// Mitsubishi GX Works2 project: Helloworlddeutrabalho   PLC: Q03UDV

PROGRAM MAIN
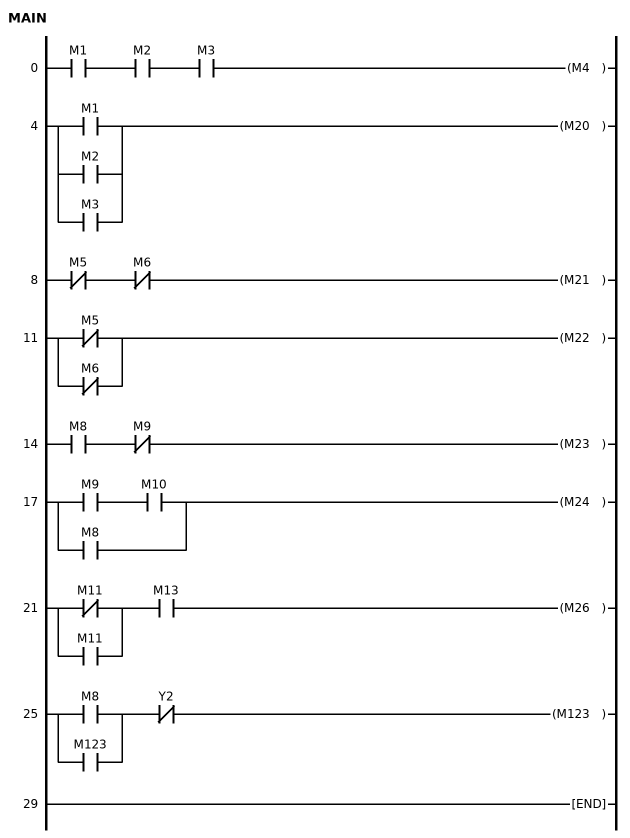
0     LD      M1
      AND     M2
      AND     M3
      OUT     M4
4     LD      M1
      OR      M2
      OR      M3
      OUT     M20
8     LDI     M5
      ANI     M6
      OUT     M21
11    LDI     M5
      ORI     M6
      OUT     M22
14    LD      M8
      ANI     M9
      OUT     M23
17    LD      M9
      AND     M10
      OR      M8
      OUT     M24
21    LDI     M11
      OR      M11
      AND     M13
      OUT     M26
25    LD      M8
      OR      M123
      ANI     Y2
      OUT     M123
29    END
END_PROGRAM
